KUKA KRL program: p01drop2_s1.src, p01drop2_s1.dat

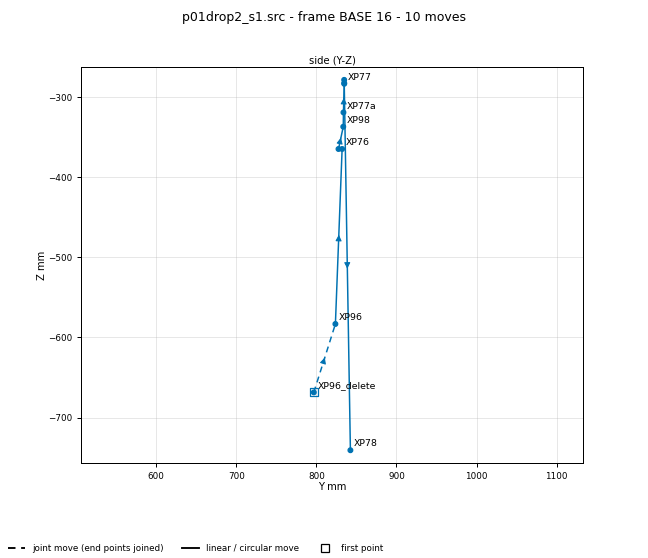
[picture p0: tool path of p01drop2_s1.src in frame BASE 16, 10 of 15 moves have a stored position in this frame; points joined in program order, loops and branches not executed]
--- p01drop2_s1.src ---
&ACCESS RVO1
&REL 4583
&PARAM TEMPLATE = C:\KRC\Roboter\Template\vorgabe
&PARAM EDITMASK = *
DEF p01drop2_s1( )

;================================================
; MODELO   : BALANCINA VIEJA
; IE GRUPO : FIP
; ESTACION : ST101
; ROBOT    : 101R1
; FUNCION  : DROP IP
;================================================

;FOLD INI
  ;FOLD BASISTECH INI
    GLOBAL INTERRUPT DECL 3 WHEN $STOPMESS==TRUE DO IR_STOPM ( )
    INTERRUPT ON 3
    BAS (#INITMOV,0 )
  ;ENDFOLD (BASISTECH INI)
;FOLD SPOTTECH INI
;USERSPOT(#INIT)
;ENDFOLD (SPOTTECH INI)
;FOLD GRIPPERTECH INI
USER_GRP(0,DUMMY,DUMMY,GDEFAULT)
INTERRUPT DECL 20 WHEN $FLAG[20]==FALSE DO GRPS(#MON_ERR,20)
;ENDFOLD (GRIPPERTECH INI)
  ;FOLD USER INI
    ;Make your modifications here

  ;ENDFOLD (USER INI)
;ENDFOLD (INI)

;ENTRAR_DEDOS()
;CERRAR_DEDOS()
;ENTRAR_RODILLO()
;ABRIR_CILINDRO_IP()
;CLAMPAR_GONDOLA()
o_type_req=FALSE

;wait position

;INICIALIZACION GRIPER

;FOLD PTP P70 Vel=100 % PDAT29 Tool[13] Base[0];%{PE}%R 5.6.13,%MKUKATPBASIS,%CMOVE,%VPTP,%P 1:PTP, 2:P70, 3:, 5:100, 7:PDAT29
$BWDSTART=FALSE
PDAT_ACT=PPDAT29
FDAT_ACT=FP70
BAS(#PTP_PARAMS,100)
PTP XP70
;ENDFOLD
;FOLD FORDTECH.Area_Req 3 Safety Position, 0 Return To Home, 0 ;%{PE}%MKUKATPUSER
;Area_Req (3,0,0)
wait for $in[19]
$out[19]=false
;ENDFOLD

;TRAYECOTORIA ENTRADA

;===========================================================
;POSICION FOTO 1 (selccionar esta linea para repetir foto 1)
;===========================================================
;FOLD OUT 38 'PETICION A DISPOSITIVO 6' State=FALSE ;%{PE}%R 5.6.13,%MKUKATPBASIS,%COUT,%VOUTX,%P 2:38, 3:PETICION A DISPOSITIVO 6, 5:FALSE, 6:
$OUT[38]=FALSE
;ENDFOLD

;FOLD PTP P97 Vel=100 % PDAT52 Tool[14]:camara Base[14]:ems_sup;%{PE}%R 5.6.13,%MKUKATPBASIS,%CMOVE,%VPTP,%P 1:PTP, 2:P97, 3:, 5:100, 7:PDAT52
$BWDSTART=FALSE
PDAT_ACT=PPDAT52
FDAT_ACT=FP97
BAS(#PTP_PARAMS,100)
PTP XP97
;ENDFOLD
;FOLD PTP P80 Vel=100 % PDAT35 Tool[14]:camara Base[14]:ems_sup;%{PE}%R 5.6.13,%MKUKATPBASIS,%CMOVE,%VPTP,%P 1:PTP, 2:P80, 3:, 5:100, 7:PDAT35
$BWDSTART=FALSE
PDAT_ACT=PPDAT35
FDAT_ACT=FP80
BAS(#PTP_PARAMS,100)
PTP XP80
;ENDFOLD


;FOLD WAIT Time=0.3 sec;%{PE}%R 5.6.13,%MKUKATPBASIS,%CWAIT,%VWAIT,%P 2:0.3
WAIT SEC 0.3
;ENDFOLD

;CHEQUEO SEÑALES RESETEADAS
MAFELEC_TECH (#CHECK_RESET, 11,0,0)

;PETICION PRIMERA FOTO
;FOLD FORDTECH.Tool_Rel 2 ;%{PE}%MKUKATPUSER
TOOL_REL (2)
;ENDFOLD

;PETICION RESULTADO FOTO
MAFELEC_TECH (#TYPE, 8,0,0)

;EVALUACION RESULTADO
SWITCH I_TYPE_INFO
CASE 2
o_type_req=FALSE
;FOLD FORDTECH.Tool_Req 2 ;%{PE}%MKUKATPUSER
TOOL_REQ (2)
;ENDFOLD
;wait for false
RECHAZOEMSINF()
goto home
case 3
o_type_req=FALSE
rechazo_bal()
GOTO HOME
ENDSWITCH

;APLICA CORRECCIONES A BASE
base_data[16]=base_data[14]
MAFELEC_TECH (#GET_CORR, 16,0,0)

tool_data[16]=tool_data[14]
;APLICA CORRECCION ANGULO A TOOL
MAFELEC_TECH (#GET_CORR_TOOL,16 ,0,0)

;REGISTRO CORRECCIONES
MAFELEC_TECH (#REG1, 11,0,0)

;FINALIZA PROCESO CORRECCIONES
o_type_req=false
wait for i_type_info==0
;FOLD FORDTECH.Tool_Req 2 ;%{PE}%MKUKATPUSER
TOOL_REQ (2)
;ENDFOLD

;POSICION SEGUNDA FOTO
xP74=xP80
;FOLD PTP P74 Vel=100 % PDAT33 Tool[16]:camara_corregida Base[16]:EMS_SUP_CORREGIDA;%{PE}%R 5.6.13,%MKUKATPBASIS,%CMOVE,%VPTP,%P 1:PTP, 2:P74, 3:, 5:100, 7:PDAT33
$BWDSTART=FALSE
PDAT_ACT=PPDAT33
FDAT_ACT=FP74
BAS(#PTP_PARAMS,100)
PTP XP74
;ENDFOLD

;FOLD WAIT Time=0.3 sec;%{PE}%R 5.6.13,%MKUKATPBASIS,%CWAIT,%VWAIT,%P 2:0.3
WAIT SEC 0.3
;ENDFOLD

;PIDE SEGUNDA FOTO
;FOLD FORDTECH.Tool_Rel 6 ;%{PE}%MKUKATPUSER
TOOL_REL (6)
;ENDFOLD

;PIDE RESULTADOS SEGUNDA FOTO
MAFELEC_TECH (#TYPE,8 ,0,0)

;EVALUA RESULTADOS FOTO
SWITCH I_TYPE_INFO
CASE 1 ;FOTO OK
o_type_req=false
wait for i_type_info==0
CASE 2
o_type_req=FALSE
;FOLD FORDTECH.Tool_Req 6 ;%{PE}%MKUKATPUSER
TOOL_REQ (6)
;ENDFOLD
RECHAZOEMSINF()
goto home
case 3
o_type_req=FALSE
rechazo_bal()
GOTO HOME
ENDSWITCH

;FINALIZA PROCESO SEGUNDA FOTO
;FOLD FORDTECH.Tool_Req 6 ;%{PE}%MKUKATPUSER
TOOL_REQ (6)
;ENDFOLD


;FOLD CHEQUEO LIMITE SEGUNDO OFFSET
;WAIT FOR EMSdownbase_OFFSETz>-200
;WAIT FOR EMSdownbase_OFFSETz<200
;WAIT FOR EMSdownbase_OFFSETx>-200
;WAIT FOR EMSdownbase_OFFSETx<200
;WAIT FOR EMSdownbase_OFFSETb>-0.400
;WAIT FOR EMSdownbase_OFFSETb<0.400
;ENDFOLD
;APLICAMOS OFFSET
;FOLD OFFSET CORR
;BASE_DATA[11].Z=EMSdownbase_CORR.Z+EMSdownbase_OFFSETz
;BASE_DATA[11].X=EMSdownbase_CORR.X+EMSdownbase_OFFSETx
;BASE_DATA[11].B=EMSdownbase_CORR.B+EMSdownbase_OFFSETb
;ENDFOLD
;goto alejandro
;SACAR_DEDOS()

if not i_dry then
;goto alejandro

;TRAYECTORIA ENTRADA A DEJAR
;FOLD PTP P96_delete Vel=100 % PDAT53 Tool[16]:camara_corregida Base[16]:EMS_SUP_CORREGIDA;%{PE}%R 5.6.13,%MKUKATPBASIS,%CMOVE,%VPTP,%P 1:PTP, 2:P96_delete, 3:, 5:100, 7:PDAT53
$BWDSTART=FALSE
PDAT_ACT=PPDAT53
FDAT_ACT=FP96_delete
BAS(#PTP_PARAMS,100)
PTP XP96_delete
;ENDFOLD
;FOLD PTP P96 Vel=100 % PDAT51 Tool[16]:camara_corregida Base[16]:EMS_SUP_CORREGIDA;%{PE}%R 5.6.13,%MKUKATPBASIS,%CMOVE,%VPTP,%P 1:PTP, 2:P96, 3:, 5:100, 7:PDAT51
$BWDSTART=FALSE
PDAT_ACT=PPDAT51
FDAT_ACT=FP96
BAS(#PTP_PARAMS,100)
PTP XP96
;ENDFOLD

;ACTIVAR TORQ MONITORING
;FOLD TORQMON SetLimits Axis 1: 40 % Axis 2: 35 % Axis 3: 35 % Axis 4: 35 % Axis 5: 40 % Axis 6: 40 %;%{PE}%R 5.6.13,%MKUKATPBASIS,%CTQ_MON,%VTQ_LIMITS,%P 2:TQ_LIMITS, 4:40, 7:35, 10:35, 13:35, 16:40, 19:40
SET_TQ_VALUES (40,35,35,35,40,40)
;ENDFOLD

;MOVIMIENTO ENTRADA A DEJAR
;FOLD LIN P76 Vel=2 m/s CPDAT14 Tool[16]:camara_corregida Base[16]:EMS_SUP_CORREGIDA;%{PE}%R 5.6.13,%MKUKATPBASIS,%CMOVE,%VLIN,%P 1:LIN, 2:P76, 3:, 5:2, 7:CPDAT14
$BWDSTART=FALSE
LDAT_ACT=LCPDAT14
FDAT_ACT=FP76
BAS(#CP_PARAMS,2)
LIN XP76
;ENDFOLD
;FOLD LIN P99 Vel=2 m/s CPDAT19 Tool[16]:camara_corregida Base[16]:EMS_SUP_CORREGIDA;%{PE}%R 5.6.13,%MKUKATPBASIS,%CMOVE,%VLIN,%P 1:LIN, 2:P99, 3:, 5:2, 7:CPDAT19
$BWDSTART=FALSE
LDAT_ACT=LCPDAT19
FDAT_ACT=FP99
BAS(#CP_PARAMS,2)
LIN XP99
;ENDFOLD
;ABRE CLAMPA
ABRIR_DEDOS()

;POSICION DEJADA

;FOLD LIN P98 Vel=2 m/s CPDAT18 Tool[16]:camara_corregida Base[16]:EMS_SUP_CORREGIDA;%{PE}%R 5.6.13,%MKUKATPBASIS,%CMOVE,%VLIN,%P 1:LIN, 2:P98, 3:, 5:2, 7:CPDAT18
$BWDSTART=FALSE
LDAT_ACT=LCPDAT18
FDAT_ACT=FP98
BAS(#CP_PARAMS,2)
LIN XP98
;ENDFOLD



;FOLD LIN P77a Vel=1 m/s CPDAT21 Tool[16]:camara_corregida Base[16]:EMS_SUP_CORREGIDA;%{PE}%R 5.6.13,%MKUKATPBASIS,%CMOVE,%VLIN,%P 1:LIN, 2:P77a, 3:, 5:1, 7:CPDAT21
$BWDSTART=FALSE
LDAT_ACT=LCPDAT21
FDAT_ACT=FP77a
BAS(#CP_PARAMS,1)
LIN XP77a
;ENDFOLD
;FOLD LIN P77 Vel=1 m/s CPDAT15 Tool[16]:camara_corregida Base[16]:EMS_SUP_CORREGIDA;%{PE}%R 5.6.13,%MKUKATPBASIS,%CMOVE,%VLIN,%P 1:LIN, 2:P77, 3:, 5:1, 7:CPDAT15
$BWDSTART=FALSE
LDAT_ACT=LCPDAT15
FDAT_ACT=FP77
BAS(#CP_PARAMS,1)
LIN XP77
;ENDFOLD
;POS FINAL ANTERIOR
;FOLD LIN p77b Vel=1 m/s CPDAT22 Tool[16]:camara_corregida Base[16]:EMS_SUP_CORREGIDA;%{PE}%R 5.6.13,%MKUKATPBASIS,%CMOVE,%VLIN,%P 1:LIN, 2:p77b, 3:, 5:1, 7:CPDAT22
$BWDSTART=FALSE
LDAT_ACT=LCPDAT22
FDAT_ACT=Fp77b
BAS(#CP_PARAMS,1)
LIN Xp77b
;ENDFOLD
;POS FINAL NUEVA
;FOLD LIN P77C Vel=1 m/s CPDAT24 Tool[16]:camara_corregida Base[16]:EMS_SUP_CORREGIDA;%{PE}%R 5.6.13,%MKUKATPBASIS,%CMOVE,%VLIN,%P 1:LIN, 2:P77C, 3:, 5:1, 7:CPDAT24
$BWDSTART=FALSE
LDAT_ACT=LCPDAT24
FDAT_ACT=FP77C
BAS(#CP_PARAMS,1)
LIN XP77C
;ENDFOLD


if not B_EMSdry then
;CIERRA CLAMPA
;clampar()
endif

;WAIT SEC 2
CERRAR_DEDOS()

if false then
;CHEQUEA CLAMPA CERRADA
endif

;FOLD WAIT Time=1 sec;%{PE}%R 5.6.13,%MKUKATPBASIS,%CWAIT,%VWAIT,%P 2:1
WAIT SEC 1
;ENDFOLD

;ESPERA RESULTADOS ACIMUT
;FOLD FORDTECH.Tool_Rel 4 ;%{PE}%MKUKATPUSER
TOOL_REL (4)
;ENDFOLD
;FOLD FORDTECH.Tool_Req 4 ;%{PE}%MKUKATPUSER
TOOL_REQ (4)
;ENDFOLD

if not B_EMSdry then
;ABRE GARRA PARA SOLTAR IP
ABRIR_CILINDRO_IP()

endif


if B_EMSdry then
;punto intermedio para liberar orejetas
endif

;MOVIMIENTO SALIDA
;FOLD LIN P78 Vel=2 m/s CPDAT16 Tool[16]:camara_corregida Base[16]:EMS_SUP_CORREGIDA;%{PE}%R 5.6.13,%MKUKATPBASIS,%CMOVE,%VLIN,%P 1:LIN, 2:P78, 3:, 5:2, 7:CPDAT16
$BWDSTART=FALSE
LDAT_ACT=LCPDAT16
FDAT_ACT=FP78
BAS(#CP_PARAMS,2)
LIN XP78
;ENDFOLD

endif
alejandro:
if i_dry then
;FOLD FORDTECH.Tool_Rel 4 ;%{PE}%MKUKATPUSER
TOOL_REL (4)
;ENDFOLD
;FOLD FORDTECH.Tool_Req 4 ;%{PE}%MKUKATPUSER
TOOL_REQ (4)
;ENDFOLD
endif

;DEJA TORQ MONITORING EN VALORES NOMINALES
;FOLD TORQMON SetDefault;%{PE}%R 5.6.13,%MKUKATPBASIS,%CTQ_MON,%VTQ_DEFAULT,%P 2:TQ_DEFAULT
SET_TQ_VALUES ( )
;ENDFOLD

;TRAYECTORIA SALIDA AREA

;wait area ems

;FOLD PTP P82 Vel=100 % PDAT37 Tool[12] Base[0];%{PE}%R 5.6.13,%MKUKATPBASIS,%CMOVE,%VPTP,%P 1:PTP, 2:P82, 3:, 5:100, 7:PDAT37
$BWDSTART=FALSE
PDAT_ACT=PPDAT37
FDAT_ACT=FP82
BAS(#PTP_PARAMS,100)
PTP XP82
;ENDFOLD




;AREA LIBRE Y TRABAJO FINALIZADO
;FOLD FORDTECH.Job_Rdy 3 , 1 ;%{PE}%MKUKATPUSER
JOB_READY (3,1)
;ENDFOLD
;FOLD FORDTECH.Area_Rel 3 ;%{PE}%MKUKATPUSER
AREA_REL (3)
;ENDFOLD

home:

END

--- p01drop2_s1.dat ---
&ACCESS RVO1
&REL 4583
&PARAM TEMPLATE = C:\KRC\Roboter\Template\vorgabe
&PARAM EDITMASK = *
DEFDAT  P01DROP2_S1
;FOLD EXTERNAL DECLARATIONS;%{PE}%MKUKATPBASIS,%CEXT,%VCOMMON,%P
;FOLD GRIPPERTECH EXT
EXT  H50 (INT  :IN,INT  :IN,INT  :IN,GRP_TYP  :IN )
;ENDFOLD (GRIPPERTECH EXT)
;FOLD SPOTTECH EXT
EXT  USERSPOT (S_COMMAND  :IN,SPOT_TYPE  :IN )
;ENDFOLD (SPOTTECH EXT)
;FOLD BASISTECH EXT;%{PE}%MKUKATPBASIS,%CEXT,%VEXT,%P
EXT  BAS (BAS_COMMAND  :IN,REAL  :IN )
DECL INT SUCCESS
;ENDFOLD (BASISTECH EXT)
;FOLD USER EXT;%{E}%MKUKATPUSER,%CEXT,%VEXT,%P
;Make here your modifications

;ENDFOLD (USER EXT)
;ENDFOLD (EXTERNAL DECLARATIONS)
DECL BASIS_SUGG_T LAST_BASIS={POINT1[] "P105                    ",POINT2[] "P105                    ",CP_PARAMS[] "CPDAT24                 ",PTP_PARAMS[] "PDAT53                  ",CONT[] "                        ",CP_VEL[] "1                       ",PTP_VEL[] "100                     ",SYNC_PARAMS[] "SYNCDAT                 ",SPL_NAME[] "S0                      "}
DECL PDAT PPDAT0={VEL 100.0,ACC 100.0,APO_DIST 100.0}
DECL E6POS XP0={X 2055.78003,Y 30.3544292,Z 1689.78503,A -75.2577133,B -0.0822966993,C 179.189499,S 2,T 3,E1 0.0,E2 0.0,E3 0.0,E4 0.0,E5 0.0,E6 0.0}
DECL FDAT FP0={TOOL_NO 0,BASE_NO 0,IPO_FRAME #BASE,POINT2[] " ",TQ_STATE FALSE}
DECL PDAT PPDAT1={VEL 100.0,ACC 100.0,APO_DIST 100.0}
DECL E6POS XP1={X -1.73297,Y 659.880615,Z 52.045929,A 0.382466912,B -0.989410281,C -2.30789709,S 2,T 3,E1 0.0,E2 0.0,E3 0.0,E4 0.0,E5 0.0,E6 0.0}
DECL FDAT FP1={TOOL_NO 3,BASE_NO 8,IPO_FRAME #BASE,POINT2[] " ",TQ_STATE FALSE}
DECL PDAT PPDAT2={VEL 100.0,ACC 100.0,APO_DIST 100.0}
DECL E6POS XP2={X 4.38160992,Y 645.864075,Z -296.583008,A 0.38227731,B -0.98957777,C -2.30757093,S 2,T 3,E1 0.0,E2 0.0,E3 0.0,E4 0.0,E5 0.0,E6 0.0}
DECL FDAT FP2={TOOL_NO 3,BASE_NO 8,IPO_FRAME #BASE,POINT2[] " ",TQ_STATE FALSE}
DECL PDAT PPDAT3={VEL 100.0,ACC 100.0,APO_DIST 100.0,APO_MODE #CPTP}
DECL E6POS XP3={X 280.11261,Y 650.938477,Z -683.81073,A 0.652623713,B 15.7282495,C -1.89291894,S 2,T 2,E1 0.0,E2 0.0,E3 0.0,E4 0.0,E5 0.0,E6 0.0}
DECL FDAT FP3={TOOL_NO 3,BASE_NO 6,IPO_FRAME #BASE,POINT2[] " ",TQ_STATE FALSE}
DECL E6POS XP4={X 2.24138999,Y 888.375122,Z -473.739807,A 0.452654511,B -1.02897203,C 1.12909102,S 2,T 11,E1 0.0,E2 0.0,E3 0.0,E4 0.0,E5 0.0,E6 0.0}
DECL FDAT FP4={TOOL_NO 10,BASE_NO 6,IPO_FRAME #BASE,POINT2[] " ",TQ_STATE FALSE}
DECL PDAT PPDAT4={VEL 100.0,ACC 100.0,APO_DIST 100.0}
DECL E6POS XP5={X 681.014282,Y 1041.89001,Z 547.901306,A 0.686961174,B -0.270723909,C -90.4319687,S 2,T 3,E1 0.0,E2 0.0,E3 0.0,E4 0.0,E5 0.0,E6 0.0}
DECL FDAT FP5={TOOL_NO 10,BASE_NO 0,IPO_FRAME #BASE,POINT2[] " ",TQ_STATE FALSE}
DECL PDAT PPDAT5={VEL 100.0,ACC 100.0,APO_DIST 100.0,APO_MODE #CPTP}
DECL LDAT LCPDAT4={VEL 2.0,ACC 100.0,APO_DIST 100.0,APO_FAC 50.0,ORI_TYP #VAR,CIRC_TYP #BASE,JERK_FAC 50.0,EXAX_IGN 0}
DECL E6POS XP6={X 368.499512,Y 715.932617,Z -549.888489,A 1.268116,B 8.31681633,C 1.09480703,S 2,T 3,E1 0.0,E2 0.0,E3 0.0,E4 0.0,E5 0.0,E6 0.0}
DECL FDAT FP6={TOOL_NO 10,BASE_NO 6,IPO_FRAME #BASE,POINT2[] " ",TQ_STATE FALSE}
DECL PDAT PPDAT6={VEL 100.0,ACC 100.0,APO_DIST 100.0,APO_MODE #CPTP}
DECL E6POS XP7={X -1.02812898,Y 658.258728,Z 11.6351805,A 0.382352501,B -0.989592195,C -2.30806804,S 2,T 3,E1 0.0,E2 0.0,E3 0.0,E4 0.0,E5 0.0,E6 0.0}
DECL FDAT FP7={TOOL_NO 3,BASE_NO 8,IPO_FRAME #BASE,POINT2[] " ",TQ_STATE FALSE}
DECL PDAT PPDAT7={VEL 100.0,ACC 100.0,APO_DIST 100.0,APO_MODE #CPTP}
DECL LDAT LCPDAT1={VEL 2.0,ACC 100.0,APO_DIST 100.0,APO_FAC 50.0,ORI_TYP #VAR,CIRC_TYP #BASE,JERK_FAC 50.0,EXAX_IGN 0}
DECL LDAT LCPDAT2={VEL 2.0,ACC 100.0,APO_DIST 100.0,APO_FAC 50.0,ORI_TYP #VAR,CIRC_TYP #BASE,JERK_FAC 50.0,EXAX_IGN 0}
DECL E6POS XP8={X 7.03343487,Y 670.851074,Z -76.543663,A 0.392349988,B -0.491735786,C 1.60772097,S 2,T 3,E1 0.0,E2 0.0,E3 0.0,E4 0.0,E5 0.0,E6 0.0}
DECL FDAT FP8={TOOL_NO 3,BASE_NO 8,IPO_FRAME #BASE,POINT2[] " ",TQ_STATE FALSE}
DECL LDAT LCPDAT3={VEL 2.0,ACC 100.0,APO_DIST 100.0,APO_FAC 50.0,ORI_TYP #VAR,CIRC_TYP #BASE,JERK_FAC 50.0,EXAX_IGN 0}
DECL LDAT LCPDAT5={VEL 2.0,ACC 100.0,APO_DIST 100.0,APO_FAC 50.0,ORI_TYP #VAR,CIRC_TYP #BASE,JERK_FAC 50.0,EXAX_IGN 0}
DECL E6POS XP9={X 3.25233507,Y 648.458984,Z -232.255203,A 0.382468998,B -0.989337206,C -2.30822897,S 2,T 3,E1 0.0,E2 0.0,E3 0.0,E4 0.0,E5 0.0,E6 0.0}
DECL FDAT FP9={TOOL_NO 3,BASE_NO 8,IPO_FRAME #BASE,POINT2[] " ",TQ_STATE FALSE}
DECL LDAT LCPDAT6={VEL 2.0,ACC 100.0,APO_DIST 100.0,APO_FAC 50.0,ORI_TYP #VAR,CIRC_TYP #BASE,JERK_FAC 50.0,EXAX_IGN 0}
DECL PDAT PPDAT8={VEL 100.0,ACC 100.0,APO_DIST 100.0,APO_MODE #CPTP}
DECL E6POS XP_11={X 557.867615,Y 658.033081,Z -559.162903,A 1.03071702,B 28.2426205,C -0.563395619,S 2,T 3,E1 0.0,E2 0.0,E3 0.0,E4 0.0,E5 0.0,E6 0.0}
DECL FDAT Fp_11={TOOL_NO 3,BASE_NO 6,IPO_FRAME #BASE,POINT2[] " ",TQ_STATE FALSE}
DECL PDAT PPDAT9={VEL 100.0,ACC 100.0,APO_DIST 100.0,APO_MODE #CPTP}
DECL PDAT PPDAT10={VEL 100.0,ACC 100.0,APO_DIST 100.0,APO_MODE #CPTP}
DECL E6POS XP_12={X 321.42569,Y 618.994995,Z -741.161377,A 1.04761398,B 14.8628902,C -1.41787004,S 2,T 2,E1 0.0,E2 0.0,E3 0.0,E4 0.0,E5 0.0,E6 0.0}
DECL FDAT Fp_12={TOOL_NO 3,BASE_NO 6,IPO_FRAME #BASE,POINT2[] " ",TQ_STATE FALSE}
DECL PDAT PPDAT11={VEL 100.0,ACC 100.0,APO_DIST 100.0,APO_MODE #CPTP}
DECL E6POS XP_13={X 203.2034,Y -117.644302,Z -811.447571,A 0.0387451202,B 6.64685392,C 0.411630988,S 2,T 2,E1 0.0,E2 0.0,E3 0.0,E4 0.0,E5 0.0,E6 0.0}
DECL FDAT Fp_13={TOOL_NO 3,BASE_NO 6,IPO_FRAME #BASE,POINT2[] " ",TQ_STATE FALSE}
DECL PDAT PPDAT12={VEL 100.0,ACC 100.0,APO_DIST 100.0,APO_MODE #CPTP}
DECL E6POS XP_14={X 5.27432823,Y 643.826782,Z -347.506897,A 0.382486194,B -0.989283502,C -2.30821395,S 2,T 3,E1 0.0,E2 0.0,E3 0.0,E4 0.0,E5 0.0,E6 0.0}
DECL FDAT Fp_14={TOOL_NO 3,BASE_NO 8,IPO_FRAME #BASE,POINT2[] " ",TQ_STATE FALSE}
DECL PDAT PPDAT13={VEL 100.0,ACC 100.0,APO_DIST 100.0,APO_MODE #CPTP}
DECL E6POS XP_15={X 5.27432823,Y 643.826782,Z -347.506897,A 0.382486194,B -0.989283502,C -2.30821395,S 2,T 3,E1 0.0,E2 0.0,E3 0.0,E4 0.0,E5 0.0,E6 0.0}
DECL FDAT Fp_15={TOOL_NO 3,BASE_NO 8,IPO_FRAME #BASE,POINT2[] " ",TQ_STATE FALSE}
DECL PDAT PPDAT14={VEL 100.0,ACC 100.0,APO_DIST 100.0,APO_MODE #CPTP}
DECL E6POS XP_16={X 698.981689,Y 1074.14404,Z 775.552124,A 1.21784198,B 0.00315639796,C -91.4702377,S 2,T 3,E1 0.0,E2 0.0,E3 0.0,E4 0.0,E5 0.0,E6 0.0}
DECL FDAT Fp_16={TOOL_NO 3,BASE_NO 0,IPO_FRAME #BASE,POINT2[] " ",TQ_STATE FALSE}
DECL PDAT PPDAT15={VEL 100.0,ACC 100.0,APO_DIST 100.0,APO_MODE #CPTP}
DECL E6POS XP_17={X 748.010376,Y 1033.51099,Z 791.128784,A -2.40130711,B -0.158479095,C -92.7849197,S 2,T 3,E1 0.0,E2 0.0,E3 0.0,E4 0.0,E5 0.0,E6 0.0}
DECL FDAT Fp_17={TOOL_NO 3,BASE_NO 0,IPO_FRAME #BASE,POINT2[] " ",TQ_STATE FALSE}
DECL PDAT PPDAT16={VEL 100.0,ACC 100.0,APO_DIST 100.0,APO_MODE #CPTP}
DECL E6POS XP_18={X 1159.33203,Y 354.279297,Z -546.946228,A 1.78119004,B 34.0756607,C 0.945991516,S 2,T 2,E1 0.0,E2 0.0,E3 0.0,E4 0.0,E5 0.0,E6 0.0}
DECL FDAT Fp_18={TOOL_NO 3,BASE_NO 6,IPO_FRAME #BASE,POINT2[] " ",TQ_STATE FALSE}
DECL PDAT PPDAT17={VEL 100.0,ACC 100.0,APO_DIST 100.0}
DECL E6POS XP_19={X -0.292107105,Y 94.9063568,Z -479.563599,A 0.452346891,B -1.029006,C 1.12948799,S 2,T 11,E1 0.0,E2 0.0,E3 0.0,E4 0.0,E5 0.0,E6 0.0}
DECL FDAT Fp_19={TOOL_NO 10,BASE_NO 11,IPO_FRAME #BASE,POINT2[] " ",TQ_STATE FALSE}
DECL PDAT PPDAT18={VEL 100.0,ACC 100.0,APO_DIST 100.0}
DECL E6POS XP_20={X 3.22195506,Y -134.998993,Z -402.318604,A 0.312464505,B -0.762871683,C -0.358684599,S 2,T 3,E1 0.0,E2 0.0,E3 0.0,E4 0.0,E5 0.0,E6 0.0}
DECL FDAT Fp_20={TOOL_NO 10,BASE_NO 11,IPO_FRAME #BASE,POINT2[] " ",TQ_STATE FALSE}
DECL PDAT PPDAT19={VEL 100.0,ACC 100.0,APO_DIST 100.0}
DECL E6POS XP_21={X -2.4641459,Y -132.361603,Z 23.9480896,A 0.312313288,B -0.762700617,C -0.358664811,S 2,T 3,E1 0.0,E2 0.0,E3 0.0,E4 0.0,E5 0.0,E6 0.0}
DECL FDAT Fp_21={TOOL_NO 10,BASE_NO 11,IPO_FRAME #BASE,POINT2[] " ",TQ_STATE FALSE}
DECL LDAT LCPDAT7={VEL 2.0,ACC 100.0,APO_DIST 100.0,APO_FAC 50.0,ORI_TYP #VAR,CIRC_TYP #BASE,JERK_FAC 50.0,EXAX_IGN 0}
DECL E6POS XP_22={X -2.82031894,Y -132.201508,Z 49.8983002,A 0.312450886,B -0.762823582,C -0.358644605,S 2,T 3,E1 0.0,E2 0.0,E3 0.0,E4 0.0,E5 0.0,E6 0.0}
DECL FDAT Fp_22={TOOL_NO 10,BASE_NO 11,IPO_FRAME #BASE,POINT2[] " ",TQ_STATE FALSE}
DECL LDAT LCPDAT8={VEL 2.0,ACC 100.0,APO_DIST 100.0,APO_FAC 50.0,ORI_TYP #VAR,CIRC_TYP #BASE,JERK_FAC 50.0,EXAX_IGN 0}
DECL E6POS XP_23={X 5.36931086,Y -136.010696,Z -564.014221,A 0.3130638,B -0.762672901,C -0.358867288,S 2,T 3,E1 0.0,E2 0.0,E3 0.0,E4 0.0,E5 0.0,E6 0.0}
DECL FDAT Fp_23={TOOL_NO 3,BASE_NO 11,IPO_FRAME #BASE,POINT2[] " ",TQ_STATE FALSE}
DECL LDAT LCPDAT9={VEL 2.0,ACC 100.0,APO_DIST 100.0,APO_FAC 50.0,ORI_TYP #VAR,CIRC_TYP #BASE,JERK_FAC 50.0,EXAX_IGN 0}
DECL E6POS XP_24={X 0.567358077,Y -135.646301,Z -275.850586,A 0.366299212,B -0.764034271,C -0.572027028,S 2,T 3,E1 0.0,E2 0.0,E3 0.0,E4 0.0,E5 0.0,E6 0.0}
DECL FDAT Fp_24={TOOL_NO 3,BASE_NO 11,IPO_FRAME #BASE,POINT2[] " ",TQ_STATE FALSE}
DECL LDAT LCPDAT10={VEL 2.0,ACC 100.0,APO_DIST 100.0,APO_FAC 50.0,ORI_TYP #VAR,CIRC_TYP #BASE,JERK_FAC 50.0,EXAX_IGN 0}
DECL E6POS XP_25={X 1210.51599,Y -154.102798,Z -591.347229,A -1.42906404,B 59.9451599,C 1.68313503,S 2,T 2,E1 0.0,E2 0.0,E3 0.0,E4 0.0,E5 0.0,E6 0.0}
DECL FDAT Fp_25={TOOL_NO 3,BASE_NO 6,IPO_FRAME #BASE,POINT2[] " ",TQ_STATE FALSE}
DECL PDAT PPDAT20={VEL 100.0,ACC 100.0,APO_DIST 100.0,APO_MODE #CPTP}
DECL E6POS XP_26={X 2094.22998,Y -533.263916,Z -1529.026,A 162.158203,B 28.4727001,C 175.247101,S 2,T 43,E1 0.0,E2 0.0,E3 0.0,E4 0.0,E5 0.0,E6 0.0}
DECL FDAT Fp_26={TOOL_NO 3,BASE_NO 6,IPO_FRAME #BASE,POINT2[] " ",TQ_STATE FALSE}
DECL PDAT PPDAT21={VEL 100.0,ACC 100.0,APO_DIST 100.0}
DECL E6POS XP_27={X 8.71923065,Y -113.524002,Z -410.962189,A 0.403023601,B -0.875886023,C 1.12987101,S 2,T 11,E1 0.0,E2 0.0,E3 0.0,E4 0.0,E5 0.0,E6 0.0}
DECL FDAT Fp_27={TOOL_NO 10,BASE_NO 11,IPO_FRAME #BASE,POINT2[] " ",TQ_STATE FALSE}
DECL PDAT PPDAT22={VEL 100.0,ACC 100.0,APO_DIST 100.0,APO_MODE #CPTP}
DECL PDAT PPDAT23={VEL 100.0,ACC 100.0,APO_DIST 100.0,APO_MODE #CPTP}
DECL E6POS XP65={X 1145.12195,Y 865.575378,Z 1562.22705,A -24.1379299,B -0.725280404,C -90.2146072,S 2,T 2,E1 0.0,E2 0.0,E3 0.0,E4 0.0,E5 0.0,E6 0.0}
DECL FDAT FP65={TOOL_NO 3,BASE_NO 0,IPO_FRAME #BASE,POINT2[] " ",TQ_STATE FALSE}
DECL PDAT PPDAT24={VEL 100.0,ACC 100.0,APO_DIST 100.0,APO_MODE #CPTP}
DECL E6POS XP66={X 1607.74902,Y 781.598511,Z 1575.47095,A -48.1744194,B -1.694278,C -88.870842,S 2,T 2,E1 0.0,E2 0.0,E3 0.0,E4 0.0,E5 0.0,E6 0.0}
DECL FDAT FP66={TOOL_NO 3,BASE_NO 0,IPO_FRAME #BASE,POINT2[] " ",TQ_STATE FALSE}
DECL PDAT PPDAT25={VEL 100.0,ACC 100.0,APO_DIST 100.0,APO_MODE #CPTP}
DECL E6POS XP67={X 2768.47705,Y 6.94654799,Z 2006.30298,A -150.0289,B 15.6658697,C -84.9255676,S 2,T 43,E1 0.0,E2 0.0,E3 0.0,E4 0.0,E5 0.0,E6 0.0}
DECL FDAT FP67={TOOL_NO 3,BASE_NO 0,IPO_FRAME #BASE,POINT2[] " ",TQ_STATE FALSE}
DECL PDAT PPDAT26={VEL 100.0,ACC 100.0,APO_DIST 100.0}
DECL E6POS XP68={X 2181.67505,Y 940.836182,Z 1193.14697,A -55.6319389,B 0.395963788,C -90.450943,S 2,T 10,E1 0.0,E2 0.0,E3 0.0,E4 0.0,E5 0.0,E6 0.0}
DECL FDAT FP68={TOOL_NO 10,BASE_NO 0,IPO_FRAME #BASE,POINT2[] " ",TQ_STATE FALSE}
DECL PDAT PPDAT27={VEL 100.0,ACC 100.0,APO_DIST 100.0,APO_MODE #CPTP}
DECL PDAT PPDAT28={VEL 100.0,ACC 100.0,APO_DIST 100.0,APO_MODE #CPTP}
DECL E6POS Xp_28={X 1159.33203,Y 354.279297,Z -546.946228,A 1.78119004,B 34.0756607,C 0.945991516,S 2,T 2,E1 0.0,E2 0.0,E3 0.0,E4 0.0,E5 0.0,E6 0.0}
DECL FDAT Fp_28={TOOL_NO 10,BASE_NO 6,IPO_FRAME #BASE,POINT2[] " ",TQ_STATE FALSE}
DECL LDAT LCPDAT11={VEL 2.0,ACC 100.0,APO_DIST 100.0,APO_FAC 50.0,ORI_TYP #VAR,CIRC_TYP #BASE,JERK_FAC 50.0,EXAX_IGN 0}
DECL E6POS Xp_29={X -2.4641459,Y -132.361603,Z 23.9480896,A 0.312313288,B -0.762700617,C -0.358664811,S 2,T 3,E1 0.0,E2 0.0,E3 0.0,E4 0.0,E5 0.0,E6 0.0}
DECL FDAT Fp_29={TOOL_NO 10,BASE_NO 11,IPO_FRAME #BASE,POINT2[] " ",TQ_STATE FALSE}
DECL E6POS XP69={X -0.110545397,Y 665.947571,Z 16.2901592,A 0.322696894,B -0.763105512,C -0.359391987,S 2,T 3,E1 0.0,E2 0.0,E3 0.0,E4 0.0,E5 0.0,E6 0.0}
DECL FDAT FP69={TOOL_NO 10,BASE_NO 8,IPO_FRAME #BASE,POINT2[] " ",TQ_STATE FALSE}
DECL LDAT LCPDAT12={VEL 2.0,ACC 100.0,APO_DIST 100.0,APO_FAC 50.0,ORI_TYP #VAR,CIRC_TYP #BASE,JERK_FAC 50.0,EXAX_IGN 0}
DECL E6POS XP70={X 704.915588,Y 2000.79797,Z 1624.86499,A -13.2152596,B 44.7332916,C 178.322906,S 2,T 11,E1 0.0,E2 0.0,E3 0.0,E4 0.0,E5 0.0,E6 0.0}
DECL FDAT FP70={TOOL_NO 13,BASE_NO 0,IPO_FRAME #BASE,POINT2[] " ",TQ_STATE FALSE}
DECL PDAT PPDAT29={VEL 100.0,ACC 100.0,APO_DIST 100.0}
DECL E6POS XP71={X 944.799622,Y -1137.30701,Z 1648.68103,A 156.109406,B 47.9737511,C 179.2742,S 2,T 10,E1 0.0,E2 0.0,E3 0.0,E4 0.0,E5 0.0,E6 0.0}
DECL FDAT FP71={TOOL_NO 0,BASE_NO 0,IPO_FRAME #BASE,POINT2[] " ",TQ_STATE FALSE}
DECL PDAT PPDAT30={VEL 100.0,ACC 100.0,APO_DIST 100.0}
DECL E6POS XP72={X 179.160904,Y 2075.0249,Z 935.252686,A -0.490047991,B 45.5180817,C 179.520294,S 2,T 11,E1 0.0,E2 0.0,E3 0.0,E4 0.0,E5 0.0,E6 0.0}
DECL FDAT FP72={TOOL_NO 0,BASE_NO 0,IPO_FRAME #BASE,POINT2[] " ",TQ_STATE FALSE}
DECL PDAT PPDAT31={VEL 100.0,ACC 100.0,APO_DIST 100.0}
DECL E6POS XP73={X -125.968903,Y 516.463684,Z -316.305115,A 90.6099472,B -1.78655696,C -0.124683701,S 2,T 10,E1 0.0,E2 0.0,E3 0.0,E4 0.0,E5 0.0,E6 0.0}
DECL FDAT FP73={TOOL_NO 8,BASE_NO 14,IPO_FRAME #BASE,POINT2[] " ",TQ_STATE FALSE}
DECL PDAT PPDAT32={VEL 100.0,ACC 100.0,APO_DIST 100.0}
DECL E6POS XP74={X -127.982498,Y 768.256714,Z -757.691406,A 89.7499771,B -0.641677022,C 0.222143695,S 2,T 11,E1 0.0,E2 0.0,E3 0.0,E4 0.0,E5 0.0,E6 0.0}
DECL FDAT FP74={TOOL_NO 16,BASE_NO 16,IPO_FRAME #BASE,POINT2[] " ",TQ_STATE FALSE}
DECL PDAT PPDAT33={VEL 100.0,ACC 100.0,APO_DIST 100.0}
DECL E6POS XP75={X 1027.97205,Y -2164.2959,Z 1001.83502,A 133.115707,B 46.7987213,C 179.862503,S 2,T 10,E1 0.0,E2 0.0,E3 0.0,E4 0.0,E5 0.0,E6 0.0}
DECL FDAT FP75={TOOL_NO 0,BASE_NO 0,IPO_FRAME #BASE,POINT2[] " ",TQ_STATE FALSE}
DECL LDAT LCPDAT13={VEL 2.0,ACC 20.0,APO_DIST 100.0,APO_FAC 50.0,ORI_TYP #VAR,CIRC_TYP #BASE,JERK_FAC 50.0,EXAX_IGN 0}
DECL E6POS XP76={X -129.740494,Y 832.164917,Z -364.766205,A 89.8703766,B -0.965562582,C 0.181317896,S 2,T 11,E1 0.0,E2 0.0,E3 0.0,E4 0.0,E5 0.0,E6 0.0}
DECL FDAT FP76={TOOL_NO 16,BASE_NO 16,IPO_FRAME #BASE,POINT2[] " ",TQ_STATE FALSE}
DECL LDAT LCPDAT14={VEL 2.0,ACC 20.0,APO_DIST 100.0,APO_FAC 50.0,ORI_TYP #VAR,CIRC_TYP #BASE,JERK_FAC 50.0,EXAX_IGN 0}
DECL E6POS XP77={X -129.478806,Y 834.796387,Z -283.402893,A 89.8703384,B -0.965359271,C 0.181190699,S 2,T 11,E1 0.0,E2 0.0,E3 0.0,E4 0.0,E5 0.0,E6 0.0}
DECL FDAT FP77={TOOL_NO 16,BASE_NO 16,IPO_FRAME #BASE,POINT2[] " ",TQ_STATE FALSE}
DECL LDAT LCPDAT15={VEL 2.0,ACC 20.0,APO_DIST 100.0,APO_FAC 50.0,ORI_TYP #VAR,CIRC_TYP #BASE,JERK_FAC 50.0,EXAX_IGN 0}
DECL E6POS XP78={X -130.945297,Y 842.500793,Z -740.850098,A 89.8722305,B -0.965318978,C 0.1806508,S 2,T 11,E1 0.0,E2 0.0,E3 0.0,E4 0.0,E5 0.0,E6 0.0}
DECL FDAT FP78={TOOL_NO 16,BASE_NO 16,IPO_FRAME #BASE,POINT2[] " ",TQ_STATE FALSE}
DECL LDAT LCPDAT16={VEL 2.0,ACC 20.0,APO_DIST 100.0,APO_FAC 50.0,ORI_TYP #VAR,CIRC_TYP #BASE,JERK_FAC 50.0,EXAX_IGN 0}
DECL E6POS XP79={X -132.875198,Y 592.144897,Z -396.872589,A 89.7520676,B -1.78774202,C 0.507864118,S 2,T 10,E1 0.0,E2 0.0,E3 0.0,E4 0.0,E5 0.0,E6 0.0}
DECL FDAT FP79={TOOL_NO 10,BASE_NO 16,IPO_FRAME #BASE,POINT2[] " ",TQ_STATE FALSE}
DECL PDAT PPDAT34={VEL 100.0,ACC 100.0,APO_DIST 100.0}
DECL E6POS XP80={X -127.982498,Y 768.256714,Z -757.691406,A 89.7499771,B -0.641677022,C 0.222143695,S 2,T 11,E1 0.0,E2 0.0,E3 0.0,E4 0.0,E5 0.0,E6 0.0}
DECL FDAT FP80={TOOL_NO 14,BASE_NO 14,IPO_FRAME #BASE,POINT2[] " ",TQ_STATE FALSE}
DECL PDAT PPDAT35={VEL 100.0,ACC 100.0,APO_DIST 100.0}
DECL E6POS XP81={X -127.982498,Y 768.256714,Z -757.691406,A 89.7499771,B -0.641677022,C 0.222143695,S 2,T 11,E1 0.0,E2 0.0,E3 0.0,E4 0.0,E5 0.0,E6 0.0}
DECL FDAT FP81={TOOL_NO 14,BASE_NO 14,IPO_FRAME #BASE,POINT2[] " ",TQ_STATE FALSE}
DECL PDAT PPDAT36={VEL 100.0,ACC 100.0,APO_DIST 100.0}
DECL PDAT PPDAT37={VEL 100.0,ACC 100.0,APO_DIST 100.0}
DECL E6POS XP82={X 704.915588,Y 2000.79797,Z 1624.86499,A -13.2152596,B 44.7332916,C 178.322906,S 2,T 11,E1 0.0,E2 0.0,E3 0.0,E4 0.0,E5 0.0,E6 0.0}
DECL FDAT FP82={TOOL_NO 12,BASE_NO 0,IPO_FRAME #BASE,POINT2[] " ",TQ_STATE FALSE}
DECL PDAT PPDAT38={VEL 100.0,ACC 100.0,APO_DIST 100.0}
DECL E6POS XP83={X 801.582214,Y 1166.55701,Z 2133.69409,A -36.2449303,B 64.0939331,C -137.098602,S 2,T 11,E1 0.0,E2 0.0,E3 0.0,E4 0.0,E5 0.0,E6 0.0}
DECL FDAT FP83={TOOL_NO 0,BASE_NO 0,IPO_FRAME #BASE,POINT2[] " ",TQ_STATE FALSE}
DECL PDAT PPDAT39={VEL 100.0,ACC 100.0,APO_DIST 100.0}
DECL E6POS XP84={X 981.520325,Y 735.968872,Z 2395.88599,A -60.3835602,B 46.7861595,C -152.051498,S 2,T 11,E1 0.0,E2 0.0,E3 0.0,E4 0.0,E5 0.0,E6 0.0}
DECL FDAT FP84={TOOL_NO 0,BASE_NO 0,IPO_FRAME #BASE,POINT2[] " ",TQ_STATE FALSE}
DECL PDAT PPDAT40={VEL 100.0,ACC 100.0,APO_DIST 100.0}
DECL E6POS XP85={X 946.800476,Y 97.3742676,Z 2526.12598,A -112.670303,B 16.4910603,C -176.548294,S 2,T 11,E1 0.0,E2 0.0,E3 0.0,E4 0.0,E5 0.0,E6 0.0}
DECL FDAT FP85={TOOL_NO 0,BASE_NO 0,IPO_FRAME #BASE,POINT2[] " ",TQ_STATE FALSE}
DECL PDAT PPDAT41={VEL 100.0,ACC 100.0,APO_DIST 100.0}
DECL E6POS XP86={X 589.351379,Y -468.337097,Z 2436.07593,A -157.786194,B 16.6084003,C -176.289505,S 2,T 10,E1 0.0,E2 0.0,E3 0.0,E4 0.0,E5 0.0,E6 0.0}
DECL FDAT FP86={TOOL_NO 0,BASE_NO 0,IPO_FRAME #BASE,POINT2[] " ",TQ_STATE FALSE}
DECL PDAT PPDAT42={VEL 100.0,ACC 100.0,APO_DIST 100.0}
DECL E6POS XP87={X 670.961914,Y -761.631775,Z 2263.86011,A -169.724503,B 10.7614298,C 171.791306,S 2,T 10,E1 0.0,E2 0.0,E3 0.0,E4 0.0,E5 0.0,E6 0.0}
DECL FDAT FP87={TOOL_NO 0,BASE_NO 0,IPO_FRAME #BASE,POINT2[] " ",TQ_STATE FALSE}
DECL PDAT PPDAT43={VEL 100.0,ACC 100.0,APO_DIST 100.0}
DECL E6POS XP88={X 364.964996,Y -1791.89001,Z 2035.68604,A -144.050598,B 66.4307404,C -139.920898,S 2,T 10,E1 0.0,E2 0.0,E3 0.0,E4 0.0,E5 0.0,E6 0.0}
DECL FDAT FP88={TOOL_NO 0,BASE_NO 0,IPO_FRAME #BASE,POINT2[] " ",TQ_STATE FALSE}
DECL PDAT PPDAT44={VEL 100.0,ACC 100.0,APO_DIST 100.0}
DECL E6POS XP89={X 364.633209,Y -1787.91199,Z 1882.00098,A -158.8311,B 69.1081772,C -155.869293,S 2,T 10,E1 0.0,E2 0.0,E3 0.0,E4 0.0,E5 0.0,E6 0.0}
DECL FDAT FP89={TOOL_NO 0,BASE_NO 0,IPO_FRAME #BASE,POINT2[] " ",TQ_STATE FALSE}
DECL PDAT PPDAT45={VEL 100.0,ACC 100.0,APO_DIST 100.0}
DECL E6POS XP90={X 801.582214,Y 1166.55701,Z 2133.69409,A -36.2449303,B 64.0939331,C -137.098602,S 2,T 11,E1 0.0,E2 0.0,E3 0.0,E4 0.0,E5 0.0,E6 0.0}
DECL FDAT FP90={TOOL_NO 0,BASE_NO 0,IPO_FRAME #BASE,POINT2[] " ",TQ_STATE FALSE}
DECL PDAT PPDAT46={VEL 100.0,ACC 100.0,APO_DIST 100.0}
DECL E6POS XP91={X 981.520325,Y 735.968872,Z 2395.88599,A -60.3835602,B 46.7861595,C -152.051498,S 2,T 11,E1 0.0,E2 0.0,E3 0.0,E4 0.0,E5 0.0,E6 0.0}
DECL FDAT FP91={TOOL_NO 0,BASE_NO 0,IPO_FRAME #BASE,POINT2[] " ",TQ_STATE FALSE}
DECL PDAT PPDAT47={VEL 100.0,ACC 100.0,APO_DIST 100.0}
DECL E6POS XP92={X 946.800476,Y 97.3742676,Z 2526.12598,A -112.670303,B 16.4910603,C -176.548294,S 2,T 11,E1 0.0,E2 0.0,E3 0.0,E4 0.0,E5 0.0,E6 0.0}
DECL FDAT FP92={TOOL_NO 0,BASE_NO 0,IPO_FRAME #BASE,POINT2[] " ",TQ_STATE FALSE}
DECL PDAT PPDAT48={VEL 100.0,ACC 100.0,APO_DIST 100.0}
DECL E6POS XP93={X 801.582214,Y 1166.55701,Z 2133.69409,A -36.2449303,B 64.0939331,C -137.098602,S 2,T 11,E1 0.0,E2 0.0,E3 0.0,E4 0.0,E5 0.0,E6 0.0}
DECL FDAT FP93={TOOL_NO 0,BASE_NO 0,IPO_FRAME #BASE,POINT2[] " ",TQ_STATE FALSE}
DECL PDAT PPDAT49={VEL 100.0,ACC 100.0,APO_DIST 100.0}
DECL E6POS XP94={X 981.520325,Y 735.968872,Z 2395.88599,A -60.3835602,B 46.7861595,C -152.051498,S 2,T 11,E1 0.0,E2 0.0,E3 0.0,E4 0.0,E5 0.0,E6 0.0}
DECL FDAT FP94={TOOL_NO 0,BASE_NO 0,IPO_FRAME #BASE,POINT2[] " ",TQ_STATE FALSE}
DECL PDAT PPDAT50={VEL 100.0,ACC 100.0,APO_DIST 100.0}
DECL E6POS XP95={X 946.800476,Y 97.3742676,Z 2526.12598,A -112.670303,B 16.4910603,C -176.548294,S 2,T 11,E1 0.0,E2 0.0,E3 0.0,E4 0.0,E5 0.0,E6 0.0}
DECL FDAT FP95={TOOL_NO 0,BASE_NO 0,IPO_FRAME #BASE,POINT2[] " ",TQ_STATE FALSE}
DECL E6POS XP96={X -127.082603,Y 823.776611,Z -583.220886,A 89.7513428,B -0.641639173,C 0.221560806,S 2,T 11,E1 0.0,E2 0.0,E3 0.0,E4 0.0,E5 0.0,E6 0.0}
DECL FDAT FP96={TOOL_NO 16,BASE_NO 16,IPO_FRAME #BASE,POINT2[] " ",TQ_STATE FALSE}
DECL PDAT PPDAT51={VEL 100.0,ACC 100.0,APO_DIST 100.0}
DECL E6POS XP97={X -74.4126129,Y 337.820313,Z -1030.99805,A 93.9724731,B -2.47263193,C 8.61725712,S 2,T 11,E1 0.0,E2 0.0,E3 0.0,E4 0.0,E5 0.0,E6 0.0}
DECL FDAT FP97={TOOL_NO 14,BASE_NO 14,IPO_FRAME #BASE,POINT2[] " ",TQ_STATE FALSE}
DECL PDAT PPDAT52={VEL 100.0,ACC 100.0,APO_DIST 100.0}
DECL E6POS XP98={X -129.302795,Y 833.587097,Z -336.985687,A 89.8949966,B -0.965553224,C 0.180301398,S 2,T 11,E1 0.0,E2 0.0,E3 0.0,E4 0.0,E5 0.0,E6 0.0}
DECL FDAT FP98={TOOL_NO 16,BASE_NO 16,IPO_FRAME #BASE,POINT2[] " ",TQ_STATE FALSE}
DECL LDAT LCPDAT18={VEL 2.0,ACC 20.0,APO_DIST 100.0,APO_FAC 50.0,ORI_TYP #VAR,CIRC_TYP #BASE,JERK_FAC 50.0,EXAX_IGN 0}
DECL E6POS XP99={X -129.790298,Y 827.635498,Z -364.774414,A 89.8709869,B -0.965503275,C 0.181457207,S 2,T 11,E1 0.0,E2 0.0,E3 0.0,E4 0.0,E5 0.0,E6 0.0}
DECL FDAT FP99={TOOL_NO 16,BASE_NO 16,IPO_FRAME #BASE,POINT2[] " ",TQ_STATE FALSE}
DECL LDAT LCPDAT19={VEL 2.0,ACC 20.0,APO_DIST 100.0,APO_FAC 50.0,ORI_TYP #VAR,CIRC_TYP #BASE,JERK_FAC 50.0,EXAX_IGN 0}
DECL PDAT PPDAT53={VEL 100.0,ACC 100.0,APO_DIST 100.0}
DECL E6POS XP100={X -127.082603,Y 823.776611,Z -583.220886,A 89.7513428,B -0.641639173,C 0.221560806,S 2,T 11,E1 0.0,E2 0.0,E3 0.0,E4 0.0,E5 0.0,E6 0.0}
DECL FDAT FP100={TOOL_NO 16,BASE_NO 16,IPO_FRAME #BASE,POINT2[] " ",TQ_STATE FALSE}
DECL E6POS XP96_delete={X -125.367897,Y 796.809814,Z -668.601685,A 89.7321472,B -0.666192114,C 0.206359804,S 2,T 11,E1 0.0,E2 0.0,E3 0.0,E4 0.0,E5 0.0,E6 0.0}
DECL FDAT FP96_delete={TOOL_NO 16,BASE_NO 16,IPO_FRAME #BASE,POINT2[] " ",TQ_STATE FALSE}
DECL LDAT LCPDAT20={VEL 2.0,ACC 20.0,APO_DIST 100.0,APO_FAC 50.0,ORI_TYP #VAR,CIRC_TYP #BASE,JERK_FAC 50.0,EXAX_IGN 0}
DECL E6POS XP101={X -128.589996,Y 827.534119,Z -283.502991,A 89.9524765,B -0.965147197,C 0.179053396,S 2,T 11,E1 0.0,E2 0.0,E3 0.0,E4 0.0,E5 0.0,E6 0.0}
DECL FDAT FP101={TOOL_NO 16,BASE_NO 16,IPO_FRAME #BASE,POINT2[] " ",TQ_STATE FALSE}
DECL E6POS XP98a={X -129.322998,Y 833.568115,Z -337.044189,A 89.8946075,B -0.96584481,C 0.181181207,S 2,T 11,E1 0.0,E2 0.0,E3 0.0,E4 0.0,E5 0.0,E6 0.0}
DECL FDAT FP98a={TOOL_NO 16,BASE_NO 16,IPO_FRAME #BASE,POINT2[] " ",TQ_STATE FALSE}
DECL LDAT LCPDAT21={VEL 2.0,ACC 20.0,APO_DIST 100.0,APO_FAC 50.0,ORI_TYP #VAR,CIRC_TYP #BASE,JERK_FAC 50.0,EXAX_IGN 0}
DECL E6POS XP102={X -129.478806,Y 834.796387,Z -283.402893,A 89.8703384,B -0.965359271,C 0.181190699,S 2,T 11,E1 0.0,E2 0.0,E3 0.0,E4 0.0,E5 0.0,E6 0.0}
DECL FDAT FP102={TOOL_NO 16,BASE_NO 16,IPO_FRAME #BASE,POINT2[] " ",TQ_STATE FALSE}
DECL E6POS XP77a={X -129.527893,Y 833.818176,Z -319.146393,A 89.8824997,B -0.967244685,C 0.177424401,S 2,T 11,E1 0.0,E2 0.0,E3 0.0,E4 0.0,E5 0.0,E6 0.0}
DECL FDAT FP77a={TOOL_NO 16,BASE_NO 16,IPO_FRAME #BASE,POINT2[] " ",TQ_STATE FALSE}
DECL LDAT LCPDAT22={VEL 2.0,ACC 20.0,APO_DIST 100.0,APO_FAC 50.0,ORI_TYP #VAR,CIRC_TYP #BASE,JERK_FAC 50.0,EXAX_IGN 0}
DECL E6POS XP103={X -129.478806,Y 834.796387,Z -283.402893,A 89.8703384,B -0.965359271,C 0.181190699,S 2,T 11,E1 0.0,E2 0.0,E3 0.0,E4 0.0,E5 0.0,E6 0.0}
DECL FDAT FP103={TOOL_NO 16,BASE_NO 16,IPO_FRAME #BASE,POINT2[] " ",TQ_STATE FALSE}
DECL E6POS Xp77b={X -129.442596,Y 834.813782,Z -282.46521,A 89.8708801,B -0.965263128,C 0.179141507,S 2,T 11,E1 0.0,E2 0.0,E3 0.0,E4 0.0,E5 0.0,E6 0.0}
DECL FDAT Fp77b={TOOL_NO 16,BASE_NO 16,IPO_FRAME #BASE,POINT2[] " ",TQ_STATE FALSE}
DECL LDAT LCPDAT23={VEL 2.0,ACC 20.0,APO_DIST 100.0,APO_FAC 50.0,ORI_TYP #VAR,CIRC_TYP #BASE,JERK_FAC 50.0,EXAX_IGN 0}
DECL E6POS XP104={X -129.442596,Y 834.813782,Z -282.46521,A 89.8708801,B -0.965263128,C 0.179141507,S 2,T 11,E1 0.0,E2 0.0,E3 0.0,E4 0.0,E5 0.0,E6 0.0}
DECL FDAT FP104={TOOL_NO 16,BASE_NO 16,IPO_FRAME #BASE,POINT2[] " ",TQ_STATE FALSE}
DECL LDAT LCPDAT24={VEL 2.0,ACC 20.0,APO_DIST 100.0,APO_FAC 50.0,ORI_TYP #VAR,CIRC_TYP #BASE,JERK_FAC 50.0,EXAX_IGN 0}
DECL E6POS XP105={X -129.442596,Y 834.813782,Z -282.46521,A 89.8708801,B -0.965263128,C 0.179141507,S 2,T 11,E1 0.0,E2 0.0,E3 0.0,E4 0.0,E5 0.0,E6 0.0}
DECL FDAT FP105={TOOL_NO 16,BASE_NO 16,IPO_FRAME #BASE,POINT2[] " ",TQ_STATE FALSE}
DECL E6POS XP77C={X -130.652603,Y 834.726379,Z -278.463013,A 89.8702927,B -0.965269923,C 0.314915687,S 2,T 11,E1 0.0,E2 0.0,E3 0.0,E4 0.0,E5 0.0,E6 0.0}
DECL FDAT FP77C={TOOL_NO 16,BASE_NO 16,IPO_FRAME #BASE,POINT2[] " ",TQ_STATE FALSE}
ENDDAT
